{attribute 'GeneratedUsingTerminal: EPP1816-0008-0016'}
{attribute addProperty BoxType "EPP1816-0008-0016"}
{attribute addProperty Description "EPP1816-0008 16 Ch. Dig. Input 24V, 10µs, D-SUB25"}
{attribute addProperty Physics "YY"}
{attribute addProperty Id "DIG_Inputs_Channel_1AT %I*DIG_Inputs_Channel_CC4551489DIG_Inputs_Channel_2AT %I*DIG_Inputs_Channel_CC4551489WcStateAT %I*WcState_9091E0EB2InfoDataAT %I*InfoData_32EB74EA10"}
{attribute addProperty CRC "1582355421"}
{attribute addProperty Size "30"}
TYPE EPP1816_5E50D3DD EXTENDS EtcSlaveBoxBase_77A0E4A7 :
STRUCT
	{attribute addProperty Name "DIG_Inputs_Channel_1"}
	DIG_Inputs_Channel_1 : DIG_Inputs_Channel_CC455148;
	{attribute addProperty Name "DIG_Inputs_Channel_2"}
	DIG_Inputs_Channel_2 : DIG_Inputs_Channel_CC455148;
	{attribute addProperty Name "WcState"}
	WcState : WcState_9091E0EB;
	{attribute addProperty Name "InfoData"}
	InfoData : InfoData_32EB74EA;
END_STRUCT
END_TYPE

(* stored: Version 1.2.0.0, ProductVersion 3.1.4024.11
   DUT EPP1816_5E50D3DD: Id {c8029eee-4b0b-413d-8390-a1ca1b5e4a21} *)
